{attribute 'qualified_only'}
VAR_GLOBAL
	
	//aCase	: ARRAY[1..3] OF ST_LAB_OuterData ;
	stCase		:	ST_LAB_CaseData; 
	stCaseFull	:	ST_LAB_CaseData; 

	
	nMax_Outers			: UINT := 50;
	nMax_Packs			: UINT := 10;


	
// 	aInputArray		: ARRAY[1..3, 1..3] OF T_MaxString := [ 
// 	['PACK01OUTER1', 'PACK02OUTER1', 'PACK03OUTER1'],
// 	['PACK01OUTER2', 'PACK02OUTER2', 'PACK03OUTER2'],
// 	['PACK01OUTER3', 'PACK02OUTER3', 'PACK03OUTER3']
// 	];


	stFBinside		: ST_FBinside;

END_VAR

(* stored: Version 1.1.0.1
   GVL GVL_test: Id {f8ade7aa-a224-4905-8a6d-e3267b15a9b2} *)
